// TwinCAT 3 PLC project LineFollowerLogic
// ProgramVersion: 3.1.4022.1
// libraries:
//   Tc2_MC2, * (Beckhoff Automation GmbH)
//   Tc2_Standard, * (Beckhoff Automation GmbH)
//   Tc2_System, * (Beckhoff Automation GmbH)
//   Tc2_Utilities, * (Beckhoff Automation GmbH)
//   Tc3_Module, * (Beckhoff Automation GmbH)
// project tree:
//   / GlobalTextList.TcGTLO, PlcTask.TcTTO, Visualization Manager.TcVMO (not stored)
//   GVLs/ GVL.TcGVL, GVL_SM.TcGVL
//   POUs/01_Simulator (SM)/ POU_SM01_LineBend.TcPOU
//   POUs/02_ScannerArray (SA)/ POU_SA01_ReadScanners.TcPOU
//   POUs/03_DriveTrain (DT)/ POU_DT01_EnableDriveTrain.TcPOU, POU_DT02_MotorControl.TcPOU
//   POUs/ MAIN.TcPOU
//   VISUs/VISUs/ Visualization.TcVIS
// real-time tasks:
//   TASK PlcTask: cycle T#10ms, priority 20, ADS port 350
// motion (NC):
//   TASK NC-DriveTrain SAF: cycle T#2ms, priority 4, ADS port 501
//   TASK NC-DriveTrain SVB: cycle T#10ms, priority 8, ADS port 511
//   AXIS LeftMotor (id 1)
//     Dynamic: Acceleration=3232.24, Deceleration=3232.24, Jerk=9696.71
//     Velo: RefSearch=21.5482368, RefSync=21.5482368, SlowManual=107.741184, FastManual=646.447104, Fast=2154.82368, Maximum=2154.82
//     OtherSettings: AllowMotionCmdToSlave=true
//     encoder EncType=1
//       EncPara: ScaleFactorNumerator=104.8576, ScaleFactorDenominator=1048576
//     drive DrvType=5
//       Analog: VeloReferenz=2370.306048, ScaleFactorActTorque=0.1
//       TimeComp: TaskDelayCycles=1
//     controller CtrType=1
//       CtrPara: PriorControlFactor=1
//         Observer: BandWidth=20
//   AXIS RightMotor (id 2)
//     OtherSettings: AllowMotionCmdToSlave=true
//     encoder EncType=1
//     drive DrvType=5
//       Analog: ScaleFactorActTorque=0.1
//       TimeComp: TaskDelayCycles=1
//     controller CtrType=1
//       CtrPara: PriorControlFactor=1
//         Observer: BandWidth=20
// I/O:
//   DEVICE Device 1 (EtherCAT Simulation), AmsNetId 10.0.0.35.2.1
//     Term 1 (EK1100) // EK1100-0000-0018
//     LeftMotorDrive (EL7211-0010) // EL7211-0010-0028
//     RightMotorDrive (EL7211-0010) // EL7211-0010-0028
// variable links:
//   LineFollowerLogic/LineFollowerLogic Instance <-> NC-DriveTrain SAF/Axes/LeftMotor
//     PlcTask Inputs/GVL.LeftMotor.NcToPlc <-> Outputs/ToPlc
//     PlcTask Outputs/GVL.LeftMotor.PlcToNc <-> Inputs/FromPlc
//   LineFollowerLogic/LineFollowerLogic Instance <-> NC-DriveTrain SAF/Axes/RightMotor
//     PlcTask Inputs/GVL.RightMotor.NcToPlc <-> Outputs/ToPlc
//     PlcTask Outputs/GVL.RightMotor.PlcToNc <-> Inputs/FromPlc

CONFIGURATION LineFollowerLogic
    RESOURCE PLC ON TwinCAT3
        TASK PlcTask(INTERVAL := T#10ms, PRIORITY := 20);
        PROGRAM MAIN WITH PlcTask : MAIN;
    END_RESOURCE
END_CONFIGURATION

// ---- GVLs/GVL.TcGVL
VAR_GLOBAL
	
	SystemON				: BOOL;
	
	LeftMotor				: AXIS_REF;
	RightMotor				: AXIS_REF;
	
	DriveTrainEnabled		: BOOL;
	
	JogLeftMotor			: BOOL;
	JogRightMotor			: BOOL;
	
	LeftLimitExceeded		: BOOL;
	RightLimitExceeded		: BOOL;
	HaltLeftMotor			: BOOL;
	HaltRightMotor			: BOOL;
	
	R100_01					: BOOL;
	R100_02					: BOOL;
	R100_03					: BOOL;
	R100_04					: BOOL;
	
END_VAR

// ---- GVLs/GVL_SM.TcGVL
VAR_GLOBAL CONSTANT
	
	LINE_ANGLE_SCALING		: REAL := 20.0;
	
END_VAR

VAR_GLOBAL
	
	LineAngle				: REAL;
	
END_VAR

// ---- POUs/MAIN.TcPOU
PROGRAM MAIN
VAR
END_VAR

POU_SM01_LineBend();

POU_SA01_ReadScanners();

POU_DT01_EnableDriveTrain();
POU_DT02_MotorControl();

END_PROGRAM

// ---- POUs/01_Simulator (SM)/POU_SM01_LineBend.TcPOU
PROGRAM POU_SM01_LineBend
VAR
END_VAR

IF LineAngle < -LINE_ANGLE_SCALING THEN
	
	R100_01 				:= TRUE;
	
ELSE
	
	R100_01					:= FALSE;
	
END_IF

IF LineAngle > LINE_ANGLE_SCALING THEN
	
	R100_04 				:= TRUE;
	
ELSE
	
	R100_04					:= FALSE;
	
END_IF

END_PROGRAM

// ---- POUs/02_ScannerArray (SA)/POU_SA01_ReadScanners.TcPOU
PROGRAM POU_SA01_ReadScanners
VAR
	
	LeftOuter				: BOOL;
	LeftInner				: BOOL; // Based on logic, could omit using inner scanners.
	RightOuter				: BOOL; // Based on logic, could omit using inner scanners.
	RightInner				: BOOL;
	
END_VAR

LeftOuter					:= R100_01;
LeftInner					:= R100_02; 
RightInner					:= R100_03; 
RightOuter					:= R100_04;

IF LeftOuter = TRUE THEN
	
	LeftLimitExceeded 		:= TRUE;
	
ELSE
	
	LeftLimitExceeded 		:= FALSE;
	
END_IF

IF RightOuter = TRUE THEN
	
	RightLimitExceeded 		:= TRUE;
	
ELSE
	
	RightLimitExceeded 		:= FALSE;
	
END_IF

END_PROGRAM

// ---- POUs/03_DriveTrain (DT)/POU_DT01_EnableDriveTrain.TcPOU
PROGRAM POU_DT01_EnableDriveTrain
VAR
	
	EnableDriveTrain 		: BOOL;
	
	fbLeftPower 			: MC_Power;
	LeftMotorEnabled		: BOOL;
	
	fbRightPower 			: MC_Power;
	RightMotorEnabled 		: BOOL;
	
END_VAR

EnableDriveTrain 			:= TRUE;

fbLeftPower(
	Axis					:= LeftMotor,
	Enable					:= EnableDriveTrain,
	Enable_Positive			:= TRUE,
	Status					=> LeftMotorEnabled);
	
fbRightPower(
	Axis					:= RightMotor,
	Enable					:= EnableDriveTrain,
	Enable_Positive			:= TRUE,
	Status					=> RightMotorEnabled);
	
IF LeftMotorEnabled AND RightMotorEnabled THEN
	
	DriveTrainEnabled 		:= TRUE;
	
ELSE
	
	DriveTrainEnabled 		:= FALSE;
	
END_IF

END_PROGRAM

// ---- POUs/03_DriveTrain (DT)/POU_DT02_MotorControl.TcPOU
PROGRAM POU_DT02_MotorControl
VAR
	
	fbHaltLeftMotor			: MC_Halt;
	fbHaltRightMotor		: MC_Halt;
	fbJogLeftMotor			: MC_Jog;
	fbJogRightMotor			: MC_Jog;
	testOnlineEdit			: BOOL;
	
END_VAR

IF NOT SystemON THEN
	
	HaltLeftMotor 			:= TRUE;
	HaltRightMotor 			:= TRUE;
	JogLeftMotor 			:= FALSE;
	JogRightMotor 			:= FALSE;
	
ELSE
	
	IF LeftLimitExceeded THEN
		
		HaltLeftMotor 		:= TRUE;
		JogLeftMotor 		:= FALSE;
		
	ELSE
		
		HaltLeftMotor 		:= FALSE;
		JogLeftMotor 		:= TRUE;
		
	END_IF
		
	IF RightLimitExceeded THEN
		
		HaltRightMotor 		:= TRUE;
		JogRightMotor 		:= FALSE;
		
	ELSE
		
		HaltRightMotor 		:= FALSE;
		JogRightMotor 		:= TRUE;
		
	END_IF
IF TRUE THEN
    testOnlineEdit			:= TRUE;
END_IF
	
END_IF

fbHaltLeftMotor(
	Axis					:= LeftMotor,
	Execute					:= HaltLeftMotor);
	
fbHaltRightMotor(
	Axis					:= RightMotor,
	Execute					:= HaltRightMotor);

fbJogLeftMotor(
	Axis					:= LeftMotor,
	JogForward				:= JogLeftMotor,
	Velocity				:= 500.0,
	Acceleration			:= 250.0,
	Deceleration			:= 500.0,
	Mode					:= E_JogMode.MC_JOGMODE_CONTINOUS);
	
fbJogRightMotor(
	Axis					:= RightMotor,
	JogForward				:= JogRightMotor,
	Velocity				:= 500.0,
	Acceleration			:= 250.0,
	Deceleration			:= 500.0,
	Mode					:= E_JogMode.MC_JOGMODE_CONTINOUS);

END_PROGRAM

// ---- GlobalTextList.TcGTLO
TEXTLIST GlobalTextList
  626 = '%10.1f'
  805 = 'Admin'
  662 = 'None'
  749 = 'Operator'
  625 = 'RotationAngle'
  359 = 'Service'
  209 = 'Turn off unit prior to Stopping runtime.'
  185 = 'Turn off unit prior to stopping runtime.'
  221 = 'Velocity\t\t\t\t:= 30.0,\n\tAcceleration\t\t\t:= 5.0,\n\tDeceleration\t\t\t:= 5.0,'
END_TEXTLIST

// ---- VISUs/VISUs/Visualization.TcVIS
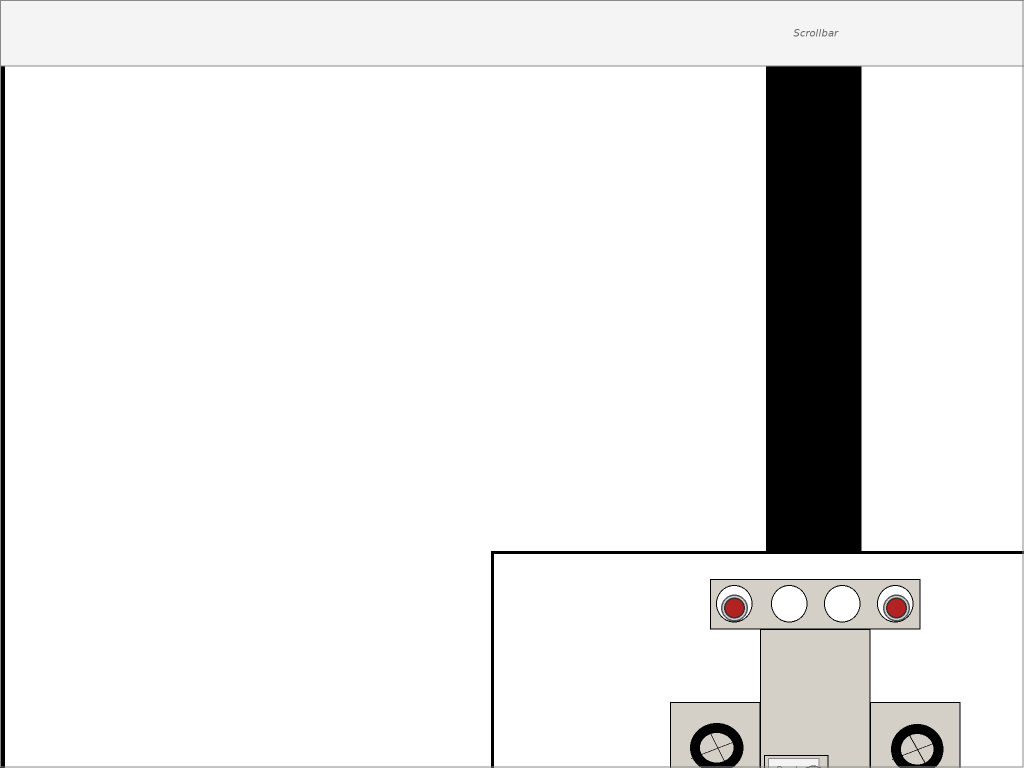
VISUALIZATION Visualization  // 1024x768
    Rectangle (0,0 1634x806)
    Rectangle (0,808 1581x618)
    Rectangle (766,-800 95x1565)
        p2858320360: LineAngle
    Rectangle (491,551 653x253)
    Group (670,579 290x221)
        Rectangle (0,123 90x90)
        Group (40,0 210x221)
            Rectangle (0,0 210x50)
            RoundedRectangle (50,50 110x171)
        Ellipse (207,6 36x37)
        Ellipse (46,6 36x37)
        Ellipse (154,6 36x37)
        Ellipse (101,6 36x37)
        Rectangle (200,123 90x90)
        Line (222,180) (271,161)
            p2858320360: POU_DT01_EnableDriveTrain.fbRightPower.Axis.NcToPlc.ActPos
        Line (21,179) (70,160)
            p2858320360: POU_DT01_EnableDriveTrain.fbLeftPower.Axis.NcToPlc.ActPos
        Ellipse (221,145 52x50)
        Ellipse (20,144 53x49)
        RoundedRectangle (94,176 64x42)
        RockerSwitch (98,179 51x37), tooltip "Turn off unit prior to Stopping runtime.", variable: SystemON, behaviour: TOGGLE, style: Switch-RockerSwitch-Gray
        Lamp1 (128,181 31x38), variable: SystemON, style: Lamp-Lamp1-Green
        Lamp1 (49,10 31x38), variable: LeftLimitExceeded, style: Lamp-Lamp1-Red
        Lamp1 (211,10 31x38), variable: RightLimitExceeded, style: Lamp-Lamp1-Red
        Line (258,189) (235,148)
            p2858320360: POU_DT01_EnableDriveTrain.fbRightPower.Axis.NcToPlc.ActPos
        Line (57,187) (37,147)
            p2858320360: POU_DT01_EnableDriveTrain.fbLeftPower.Axis.NcToPlc.ActPos
    Scrollbar (0,0 1632x66)
        p3598130195: -50
        p1057716461: LineAngle
    Meter180 (1235,461 250x250), value: LeftMotor.NcToPlc.ActVelo, style: Meter-Meter180-Gray, scale format: %.1f, scale 0..100
    BarDisplayImage (1207,652 300x50), value: RightMotor.NcToPlc.ActVelo, style: BarDisplayImage-Gray, scale format: %.1f, scale 0..100
END_VISUALIZATION
